% RSLogix 500 project Job 12 Part 1 - Leo Kniffen.RSS, saved by version 10.00.00.00 %
PROJECT "ML04B"    % processor: Bul.1763 MicroLogix 1100 Series B %

PROGRAM FILES
  LAD 2   8 rungs

DATA FILES
  O0 OUTPUT  4 elements
  I1 INPUT  6 elements
  S2 STATUS  66 elements
  B3 BINARY  1 elements
  T4 TIMER  1 elements
  C5 COUNTER  1 elements
  R6 CONTROL  1 elements
  N7 INTEGER  1 elements
  F8 FLOAT  1 elements

LADDER 2
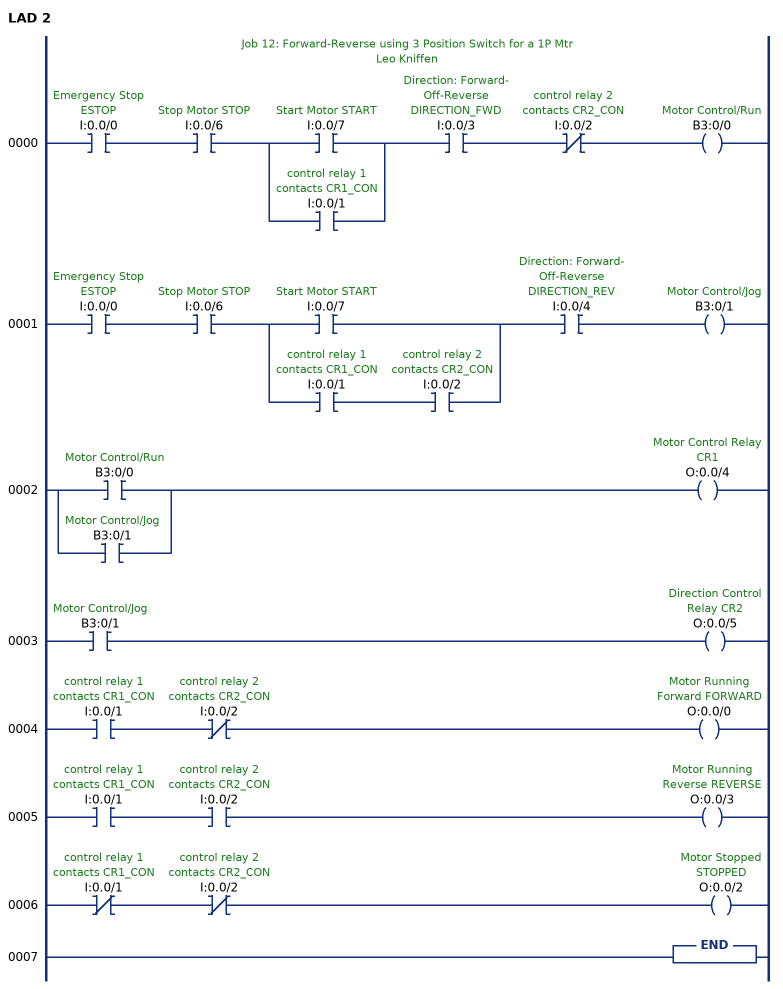
% Rung: 0 %
% Job 12: Forward-Reverse using 3 Position Switch for a 1P Mtr
% Leo Kniffen %
SOR XIC I:0.0/0 XIC I:0.0/6 BST XIC I:0.0/7 NXB XIC I:0.0/1 BND XIC I:0.0/3 XIO I:0.0/2 OTE B3:0/0 EOR
%   I:0.0/0  ESTOP  "Emergency Stop" %
%   I:0.0/6  STOP  "Stop Motor" %
%   I:0.0/7  START  "Start Motor" %
%   I:0.0/1  CR1_CON  "control relay 1 contacts" %
%   I:0.0/3  DIRECTION_FWD  "Direction: Forward- Off-Reverse" %
%   I:0.0/2  CR2_CON  "control relay 2 contacts" %
%   B3:0/0  "Motor Control/Run" %
% Rung: 1 %
SOR XIC I:0.0/0 XIC I:0.0/6 BST XIC I:0.0/7 NXB XIC I:0.0/1 XIC I:0.0/2 BND XIC I:0.0/4 OTE B3:0/1 EOR
%   I:0.0/0  ESTOP  "Emergency Stop" %
%   I:0.0/6  STOP  "Stop Motor" %
%   I:0.0/7  START  "Start Motor" %
%   I:0.0/1  CR1_CON  "control relay 1 contacts" %
%   I:0.0/2  CR2_CON  "control relay 2 contacts" %
%   I:0.0/4  DIRECTION_REV  "Direction: Forward- Off-Reverse" %
%   B3:0/1  "Motor Control/Jog" %
% Rung: 2 %
SOR BST XIC B3:0/0 NXB XIC B3:0/1 BND OTE O:0.0/4 EOR
%   B3:0/0  "Motor Control/Run" %
%   B3:0/1  "Motor Control/Jog" %
%   O:0.0/4  CR1  "Motor Control Relay" %
% Rung: 3 %
SOR XIC B3:0/1 OTE O:0.0/5 EOR
%   B3:0/1  "Motor Control/Jog" %
%   O:0.0/5  CR2  "Direction Control Relay" %
% Rung: 4 %
SOR XIC I:0.0/1 XIO I:0.0/2 OTE O:0.0/0 EOR
%   I:0.0/1  CR1_CON  "control relay 1 contacts" %
%   I:0.0/2  CR2_CON  "control relay 2 contacts" %
%   O:0.0/0  FORWARD  "Motor Running Forward" %
% Rung: 5 %
SOR XIC I:0.0/1 XIC I:0.0/2 OTE O:0.0/3 EOR
%   I:0.0/1  CR1_CON  "control relay 1 contacts" %
%   I:0.0/2  CR2_CON  "control relay 2 contacts" %
%   O:0.0/3  REVERSE  "Motor Running Reverse" %
% Rung: 6 %
SOR XIO I:0.0/1 XIO I:0.0/2 OTE O:0.0/2 EOR
%   I:0.0/1  CR1_CON  "control relay 1 contacts" %
%   I:0.0/2  CR2_CON  "control relay 2 contacts" %
%   O:0.0/2  STOPPED  "Motor Stopped" %
% Rung: 7 %
SOR END EOR

OTHER DOCUMENTED ADDRESSES
  I:0.0/5  RUN_JOG  "Run/Jog Mode (A=Run, B=Jog)"
  I:0.0/8  JOG  "Jog Motor"
  O:0.0/1  YEL_L  "yellow light"
